{attribute addProperty BoxType "EP4314-1002-0016"}
{attribute addProperty Id "DI_InputsAT %I*DI_Inputs_ECDEFC7F3240AI_Standard_ChannelAT %I*ARRAY[0..1] OF AI_Standard_Channel_F16A160D6480AO_Standard_ChannelAT %Q*ARRAY[0..1] OF AO_Standard_Channel_F57FA4F93240WcStateAT %I*WcState_F855686C1620InfoDataAT %I*InfoData_BC63D37F80100"}
{attribute addProperty CRC "438355800"}
{attribute addProperty SizeInBites "224"}
{attribute addProperty SizeInBytes "28"}
TYPE EP4314_43F10CD1 :
STRUCT
	{attribute addProperty Name "DI_Inputs"}
	DI_Inputs : DI_Inputs_ECDEFC7F;
	{attribute addProperty Name "AI_Standard_Channel"}
	AI_Standard_Channel : ARRAY[0..1] OF AI_Standard_Channel_F16A160D;
	{attribute addProperty Name "AO_Standard_Channel"}
	AO_Standard_Channel : ARRAY[0..1] OF AO_Standard_Channel_F57FA4F9;
	{attribute addProperty Name "WcState"}
	WcState : WcState_F855686C;
	{attribute addProperty Name "InfoData"}
	InfoData : InfoData_BC63D37F;
END_STRUCT
END_TYPE

(* stored: Version 1.2.0.0, ProductVersion 3.1.4024.9
   DUT EP4314_43F10CD1: Id {dd09cedc-6b71-4498-bcb1-06ebdb960e60} *)
